PROGRAM MAIN
VAR
END_VAR

END_PROGRAM

(* stored: Version 1.1.0.1
   POU MAIN: Id {d33ae895-c531-48a2-b7d5-2b28e3a1d85b} *)
